(* Schneider Machine Expert - Basic project 撞击便携一体机, file version 1.5.0.0 *)
(* ProjectInformations: Name=New project *)

HARDWARE
  Cpu 0: TM200CE24U
  Cartridge1 0: TMCR2AM3
  EthernetConfiguration: NetworkName=M200, IpAllocationMode=FixedAddress, IpAddress=0.0.0.0, SubnetMask=0.0.0.0
  EthernetConfiguration: NetworkName=M221, IpAllocationMode=FixedAddress, IpAddress=0.0.0.0, SubnetMask=0.0.0.0
  SerialLineConfiguration: Baud=Baud19200, Parity=ParityEven, DataBits=DataBits8, StopBits=StopBits1, PhysicalMedium=PhysicalMediumRs485, TransmissionMode=TransmissionModeModbusRtu, SlaveId=1, Addressing=SlaveAddressing
  MastTask: UsePeriodScanMode=false, PeriodScan=2
  FastTask: Period=255
  CpuBehavior: StartingMode=StartAsPreviousState, AutoSaveRamOnEeprom=true, WatchdogPeriod=250

SYMBOLS  (address, symbol, comment, settings)
  %M0         "步进电机使能"
  %M1         "步进电机就位"
  %M2         "步进电机正向限位"
  %M3         "步进电机反向限位"
  %M4         "自动升锤任务表启动"
  %M5         "自动升锤任务表循环执行"
  %M6         "自动升锤任务表暂停执行"
  %M7         "装药任务表启动"
  %M8         "装药任务表循环执行"
  %M9         "装药任务表暂停执行"
  %M10        "吸放重锤电磁铁得电指令"
  %M11        "吸放重锤电磁铁失电指令"
  %M12        "自动降锤任务表启动"
  %M13        "落锤运动停止"
  %M15        "步进电机指令复位"
  %M16        "落锤运动模式(自动=1,手动=0)"
  %M17        "手动升锤"
  %M18        "手动降锤"
  %M19        "步进电机复位后n秒"
  %M20        "加压电机后退指令"
  %M21        "加压电机前进指令"
  %M22        "加压电机停止指令"
  %M23        "步进电机报警状态位"
  %M24        "系统复位"
  %M25        "撞击摩擦控制工艺区分位"
  %M26        "装药加压电机后退末程"
  %M30        "上位机重锤释放指令"
  %M31        "加压完成"
  %M32        "压力传感器开始受压时"
  %M33        "压力值接近设定压力时"
  %M34        "上位机装药指令"
  %M35        "靠近落锤位"
  %M36        "到达最低位"
  %M37        "到达装药位"
  %M38        "装药完成"
  %M39        "落锤运动方向位"
  %M40        "落锤向上减速位"
  %M41        "落锤向下减速位"
  %M42        "落锤向上运动到位"
  %M43        "落锤向下运动到位"
  %M45        "落锤运动到位"
  %M46        "落锤释放完成"
  %S13      SB_FIRSTRUN  "Indicates the first controller cycle in RUN mode"
  %MW1        "重锤位移中间原始值"
  %MW2        "重锤位移数字量差值"
  %MW3        "加压压力中间原始值"
  %MW4        "加压压力数字量差值"
  %MW5        "上位机落锤高度设置值(精确度：0.1mm)"
  %MW6        "上位机加压压力设置值(精确度:0.01T)"
  %MW7        "上位机重锤高度显示值（精确度：0.1mm)"
  %MW8        "上位机加压压力显示值(精确度:0.01T)"
  %MW9        "重锤运动量程值(精确度：0.1mm)"
  %MW10       "上位机高度显示中间值"
  %MW12       "上位机压力显示中间值"
  %MW15       "加压压力实数差值"
  %MW17       "加压压力实际实数值(单位:T)"
  %MW19       "重锤运动量程中间值"
  %MW21       "重锤位移实数差值"
  %MW23       "重锤位移实际实数值"
  %MW25       "重锤运动量程值"
  %MW27       "重锤相对位移实数值"
  %MW30       "上位机加压设置中间值"
  %MW32       "上位机加压设置转换值"
  %MW34       "加压电机频率设置值"
  %MW36       "加压电机频率设置值与量程比值"
  %MW38       "加压电机频率设置值对应数字量差值"
  %MW40       "加压电机频率设置值对应数字量值"
  %MW42       "加压电机频率整数值"
  %MW45       "加压设定值靠近值"
  %MW47       "上位机高度设置中间值"
  %MW49       "上位机高度设置转换值"
  %MW51       "落锤上升减速位移值"
  %MW53       "落锤下降减速位移值"
  %MW55       "位移相对值"
  %TM0        [Type=TP, Preset=1, Base=OneSecond]
  %TM1        [Preset=15, Base=OneHundredMilliSeconds]
  %TM2        [Preset=10, Base=OneSecond]
  %TM3        [Preset=21, Base=OneSecond]
  %TM4        [Preset=1, Base=OneSecond]
  %TM5        [Type=TP, Preset=2, Base=OneSecond]
  %MC_MOTIONTASK_PTO0   "升锤"  [Axis(Value(PtoAxis=PTO0)), StartStep(Value(int=1)), EndStep(Value(int=3)), Table(Value(PtoMotionTaskTable=Mt0))]
  %MC_MOTIONTASK_PTO1   "装药"  [Axis(Value(PtoAxis=PTO0)), StartStep(Value(int=1)), EndStep(Value(int=5)), Table(Value(PtoMotionTaskTable=Mt1))]
  %MC_MOVEABS_PTO0 绝对位置任务  [Axis(Value(PtoAxis=None)), Position(Value(int=10000)), Velocity(Value(int=20000)), Acceleration(Value(int=1000)), Deceleration(Value(int=1000)), JerkRatio(Value(int=0)), BufferMode(Value(BufferMode=McAborting))]
  %MC_MOVEREL_PTO1 相对位置任务1  [Axis(Value(PtoAxis=None)), Distance(Value(int=10000)), Velocity(Value(int=320)), Acceleration(Value(int=30)), Deceleration(Value(int=30)), JerkRatio(Value(int=0)), BufferMode(Value(BufferMode=McAborting))]
  %MC_MOVEREL_PTO6   [Axis(Value(PtoAxis=PTO0)), Distance(Value(int=10000)), Velocity(Value(int=200)), Acceleration(Value(int=30)), Deceleration(Value(int=30)), JerkRatio(Value(int=0)), BufferMode(Value(BufferMode=McAborting))]
  %MC_MOVEREL_PTO7   [Axis(Value(PtoAxis=PTO0)), Distance(Value(int=-10000)), Velocity(Value(int=50)), Acceleration(Value(int=30)), Deceleration(Value(int=30)), JerkRatio(Value(int=0)), BufferMode(Value(BufferMode=McAborting))]
  %MC_MOVEREL_PTO8   [Axis(Value(PtoAxis=PTO0)), Distance(Value(int=10000)), Velocity(Value(int=50)), Acceleration(Value(int=30)), Deceleration(Value(int=30)), JerkRatio(Value(int=0)), BufferMode(Value(BufferMode=McAborting))]
  %MC_MOVEVEL_PTO0 速度任务  [Axis(Value(PtoAxis=None)), Velocity(Value(int=10000)), Acceleration(Value(int=100)), Deceleration(Value(int=1000)), JerkRatio(Value(int=0)), Direction(Value(Direction=McPositiveDirection)), BufferMode(Value(BufferMode=McAborting))]
  %MC_POWER_PTO0   [Axis(Value(PtoAxis=PTO0))]
  %MC_RESET_PTO0   [Axis(Value(PtoAxis=PTO0))]
  %MC_SETPOS_PTO0 位置设定  [Axis(Value(PtoAxis=None)), Position(Value(int=0))]
  %MC_STOP_PTO0   [Axis(Value(PtoAxis=PTO0)), Deceleration(Value(int=30)), JerkRatio(Value(int=0))]
  %MT0        "升锤"  [IsConfigured=true, MotionSteps(MotionStep(Step=12, Type=None, Next=Done, Delay=0), MotionStep(Step=11, Type=None, Next=Done, Delay=0), MotionStep(Step=10, Type=None, Next=Done, Delay=0), MotionStep(Step=1, Pto=%MC_MOVEREL_PTO0, Type=MoveRelative, Next=SwEvent, Delay=0, Event=%M40), MotionStep(Step=13, Type=None, Next=Done, Delay=0), MotionStep(Step=2, Pto=%MC_MOVEREL_PTO5, Type=MoveRelative, Next=]
  %MT1        "装药"  [IsConfigured=true, MotionSteps(MotionStep(Step=1, Pto=%MC_MOVEREL_PTO1, Type=MoveRelative, Next=SwEvent, Delay=0, Event=%M35), MotionStep(Step=3, Pto=%MC_HALT_PTO1, Type=Halt, Next=Delay, Delay=500), MotionStep(Step=4, Pto=%MC_MOVEREL_PTO4, Type=MoveRelative, Next=SwEvent, Delay=0, Event=%M37), MotionStep(Step=5, Pto=%MC_HALT_PTO3, Type=Halt, Next=Done, Delay=0), MotionStep(Step=6, Type=None, Next]
  %I0.0       "加压电机后退限位"
  %I0.1       "安全门开关"
  %Q0.0       "步进电机脉冲位"
  %Q0.1       "吸放重锤电磁铁"
  %Q0.2       "步进电机方向位"
  %Q0.3       "加压电机后退"
  %Q0.4       "加压电机前进"
  %IW0.100  重锤原始位移值  [Type=Type_4_20_mA, Scope=Scope_Normal, Minimum=4000, Maximum=20000]
  %IW0.101  加压原始压力值  [Type=Type_4_20_mA, Scope=Scope_Normal, Minimum=4000, Maximum=20000]
  %QW0.100  加压变频电机频率  [Type=Type_4_20_mA, Scope=Scope_Normal, Minimum=4000, Maximum=20000]

POU 步进电机
  (* SectionNumber=1, IsGrafcet=false *)

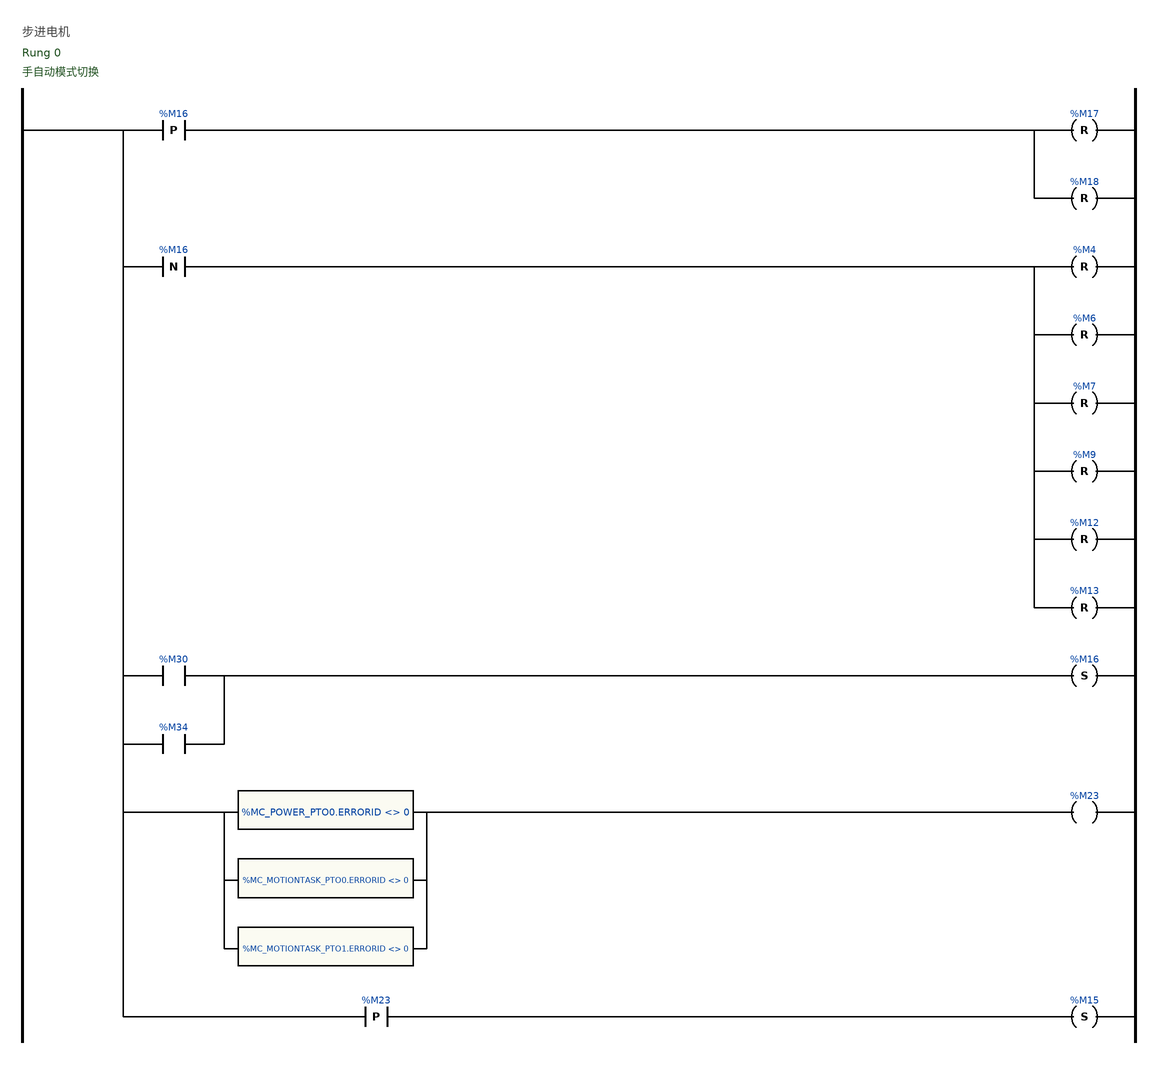

// Rung 0
// 手自动模式切换
  LD 1
  MPS
  ANDR %M16
  R %M17
  R %M18
  MRD
  ANDF %M16
  R %M4
  R %M6
  R %M7
  R %M9
  R %M12
  R %M13
  MRD
  AND( %M30
  OR %M34
  )
  S %M16
  MRD
  AND( [ %MC_POWER_PTO0.ERRORID <> 0 ]
  OR( [ %MC_MOTIONTASK_PTO0.ERRORID <> 0 ]
  OR [ %MC_MOTIONTASK_PTO1.ERRORID <> 0 ]
  )
  )
  ST %M23
  MPP
  ANDR %M23
  S %M15
  // as ST:
  //   IF RISING(%M16) THEN %M17 := FALSE; END_IF;
  //   IF RISING(%M16) THEN %M18 := FALSE; END_IF;
  //   IF FALLING(%M16) THEN %M4 := FALSE; END_IF;
  //   IF FALLING(%M16) THEN %M6 := FALSE; END_IF;
  //   IF FALLING(%M16) THEN %M7 := FALSE; END_IF;
  //   IF FALLING(%M16) THEN %M9 := FALSE; END_IF;
  //   IF FALLING(%M16) THEN %M12 := FALSE; END_IF;
  //   IF FALLING(%M16) THEN %M13 := FALSE; END_IF;
  //   IF %M30 OR %M34 THEN %M16 := TRUE; END_IF;
  //   %M23 := %MC_POWER_PTO0.ERRORID <> 0 OR %MC_MOTIONTASK_PTO0.ERRORID <> 0 OR %MC_MOTIONTASK_PTO1.ERRORID <> 0;
  //   IF RISING(%M23) THEN %M15 := TRUE; END_IF;

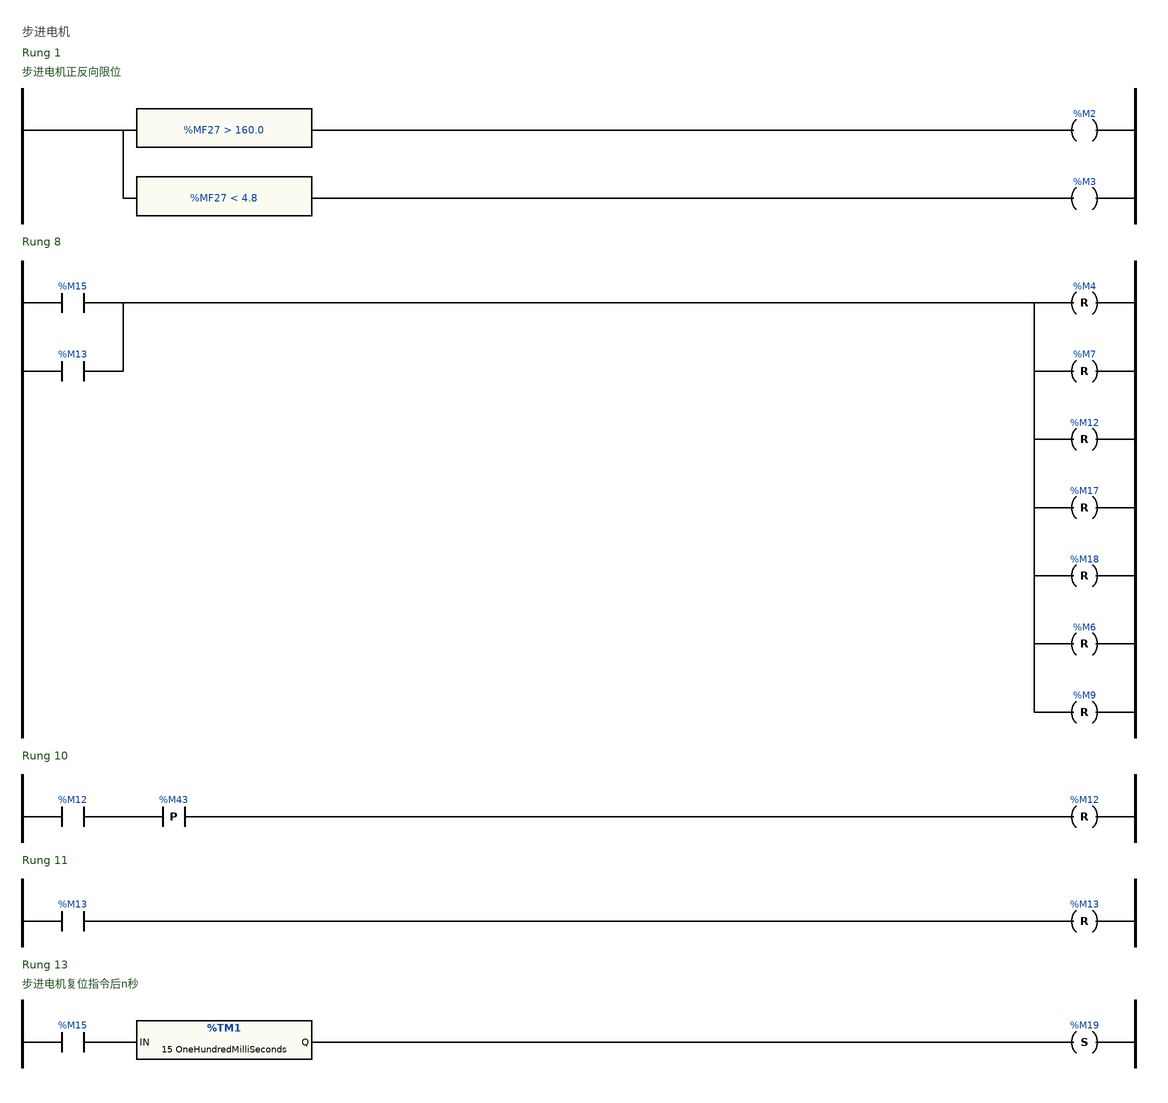

// Rung 1
// 步进电机正反向限位
  LD 1
  MPS
  AND [ %MF27 > 160.0 ]
  ST %M2
  MPP
  AND [ %MF27 < 4.8 ]
  ST %M3
  // as ST:
  //   %M2 := %MF27 > 160.0;
  //   %M3 := %MF27 < 4.8;

// Rung 2
// 步进电机使能及准备就位
  BLK %MC_POWER_PTO0
  LDN %M0
  Enable
  LDN %M1
  DriveReady
  LDN %M2
  OR %M15
  LimP
  LDN %M3
  OR %M15
  LimN
  END_BLK
  // as ST:
  //   %MC_POWER_PTO0(ENABLE := NOT %M0, DRIVEREADY := NOT %M1, LIMP := NOT %M2 OR %M15, LIMN := NOT %M3 OR %M15);
  (* the ladder stored for this rung does not match its IL; not drawn *)

// Rung 3
// 自动升锤
  BLK %MC_MOTIONTASK_PTO0
  LD %M4
  ANDN %M12
  ANDN %M7
  AND %M16
  Start
  LD %M5
  Loop
  LD %M6
  Pause
  OUT_BLK
  LD Ended
  R %M4
  END_BLK
  // as ST:
  //   %MC_MOTIONTASK_PTO0(START := %M4 AND NOT %M12 AND NOT %M7 AND %M16, LOOP := %M5, PAUSE := %M6);
  //   IF %MC_MOTIONTASK_PTO0.Ended THEN %M4 := FALSE; END_IF;
  (* the ladder stored for this rung does not match its IL; not drawn *)

// Rung 4
// 自动装药
  BLK %MC_MOTIONTASK_PTO1
  LD %M7
  ANDN %M4
  ANDN %M12
  AND %M16
  Start
  LD %M8
  Loop
  LD %M9
  Pause
  OUT_BLK
  LD Ended
  R %M7
  S %M38
  END_BLK
  // as ST:
  //   %MC_MOTIONTASK_PTO1(START := %M7 AND NOT %M4 AND NOT %M12 AND %M16, LOOP := %M8, PAUSE := %M9);
  //   IF %MC_MOTIONTASK_PTO1.Ended THEN %M7 := FALSE; END_IF;
  //   IF %MC_MOTIONTASK_PTO1.Ended THEN %M38 := TRUE; END_IF;
  (* the ladder stored for this rung does not match its IL; not drawn *)

// Rung 5
// 自动降锤
  BLK %MC_MOVEREL_PTO6
  LD %M12
  ANDN %M4
  ANDN %M7
  AND %M16
  Execute
  END_BLK
  // as ST:
  //   %MC_MOVEREL_PTO6(EXECUTE := %M12 AND NOT %M4 AND NOT %M7 AND %M16);
  (* the ladder stored for this rung does not match its IL; not drawn *)

// Rung 6
// 手动升锤
  BLK %MC_MOVEREL_PTO7
  LD %M17
  ANDN %M18
  ANDN %M16
  OR( %M19
  AND %M3
  )
  Execute
  END_BLK
  // as ST:
  //   %MC_MOVEREL_PTO7(EXECUTE := %M17 AND NOT %M18 AND NOT %M16 OR %M19 AND %M3);
  (* the ladder stored for this rung does not match its IL; not drawn *)

// Rung 7
// 手动降锤
  BLK %MC_MOVEREL_PTO8
  LD %M18
  ANDN %M17
  ANDN %M16
  OR( %M19
  AND %M2
  )
  Execute
  END_BLK
  // as ST:
  //   %MC_MOVEREL_PTO8(EXECUTE := %M18 AND NOT %M17 AND NOT %M16 OR %M19 AND %M2);
  (* the ladder stored for this rung does not match its IL; not drawn *)

// Rung 8
  LD %M15
  OR %M13
  R %M4
  R %M7
  R %M12
  R %M17
  R %M18
  R %M6
  R %M9
  // as ST:
  //   IF %M15 OR %M13 THEN %M4 := FALSE; END_IF;
  //   IF %M15 OR %M13 THEN %M7 := FALSE; END_IF;
  //   IF %M15 OR %M13 THEN %M12 := FALSE; END_IF;
  //   IF %M15 OR %M13 THEN %M17 := FALSE; END_IF;
  //   IF %M15 OR %M13 THEN %M18 := FALSE; END_IF;
  //   IF %M15 OR %M13 THEN %M6 := FALSE; END_IF;
  //   IF %M15 OR %M13 THEN %M9 := FALSE; END_IF;

// Rung 9
  BLK %MC_STOP_PTO0
  LD %M15
  OR( %M12
  ANDR %M43
  )
  OR %M13
  OR %M19
  Execute
  END_BLK
  // as ST:
  //   %MC_STOP_PTO0(EXECUTE := %M15 OR %M12 AND RISING(%M43) OR %M13 OR %M19);
  (* the ladder stored for this rung does not match its IL; not drawn *)

// Rung 10
  LD %M12
  ANDR %M43
  R %M12
  // as ST:
  //   IF %M12 AND RISING(%M43) THEN %M12 := FALSE; END_IF;

// Rung 11
  LD %M13
  R %M13
  // as ST:
  //   IF %M13 THEN %M13 := FALSE; END_IF;

// Rung 12
  BLK %MC_RESET_PTO0
  LD %M15
  Execute
  END_BLK
  // as ST:
  //   %MC_RESET_PTO0(EXECUTE := %M15);
  (* the ladder stored for this rung does not match its IL; not drawn *)

// Rung 13
// 步进电机复位指令后n秒
  BLK %TM1
  LD %M15
  IN
  OUT_BLK
  LD Q
  S %M19
  END_BLK
  // as ST:
  //   %TM1(IN := %M15);
  //   IF %TM1.Q THEN %M19 := TRUE; END_IF;

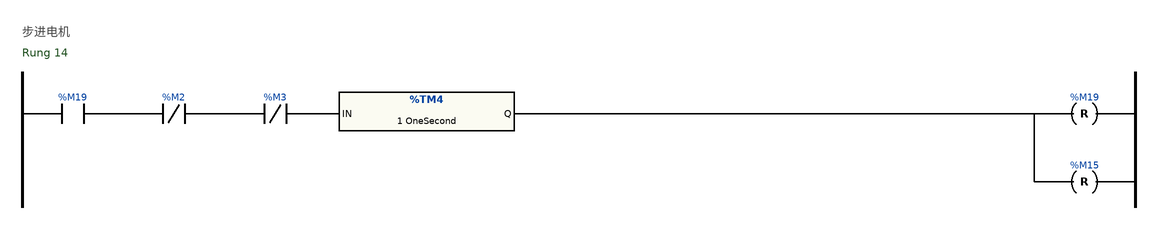

// Rung 14
  BLK %TM4
  LD %M19
  ANDN %M2
  ANDN %M3
  IN
  OUT_BLK
  LD Q
  R %M19
  R %M15
  END_BLK
  // as ST:
  //   %TM4(IN := %M19 AND NOT %M2 AND NOT %M3);
  //   IF %TM4.Q THEN %M19 := FALSE; END_IF;
  //   IF %TM4.Q THEN %M15 := FALSE; END_IF;

POU 吸放重锤电磁铁
  (* SectionNumber=2, IsGrafcet=false *)

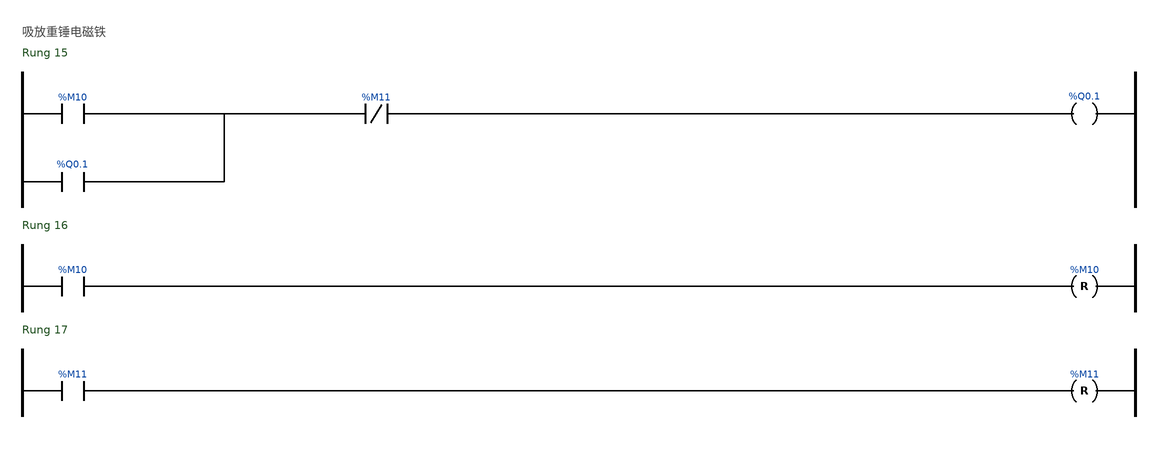

// Rung 15
  LD %M10
  OR %Q0.1
  ANDN %M11
  ST %Q0.1
  // as ST:
  //   %Q0.1 := (%M10 OR %Q0.1) AND NOT %M11;

// Rung 16
  LD %M10
  R %M10
  // as ST:
  //   IF %M10 THEN %M10 := FALSE; END_IF;

// Rung 17
  LD %M11
  R %M11
  // as ST:
  //   IF %M11 THEN %M11 := FALSE; END_IF;

POU 变频加压电机
  (* SectionNumber=3, IsGrafcet=false *)

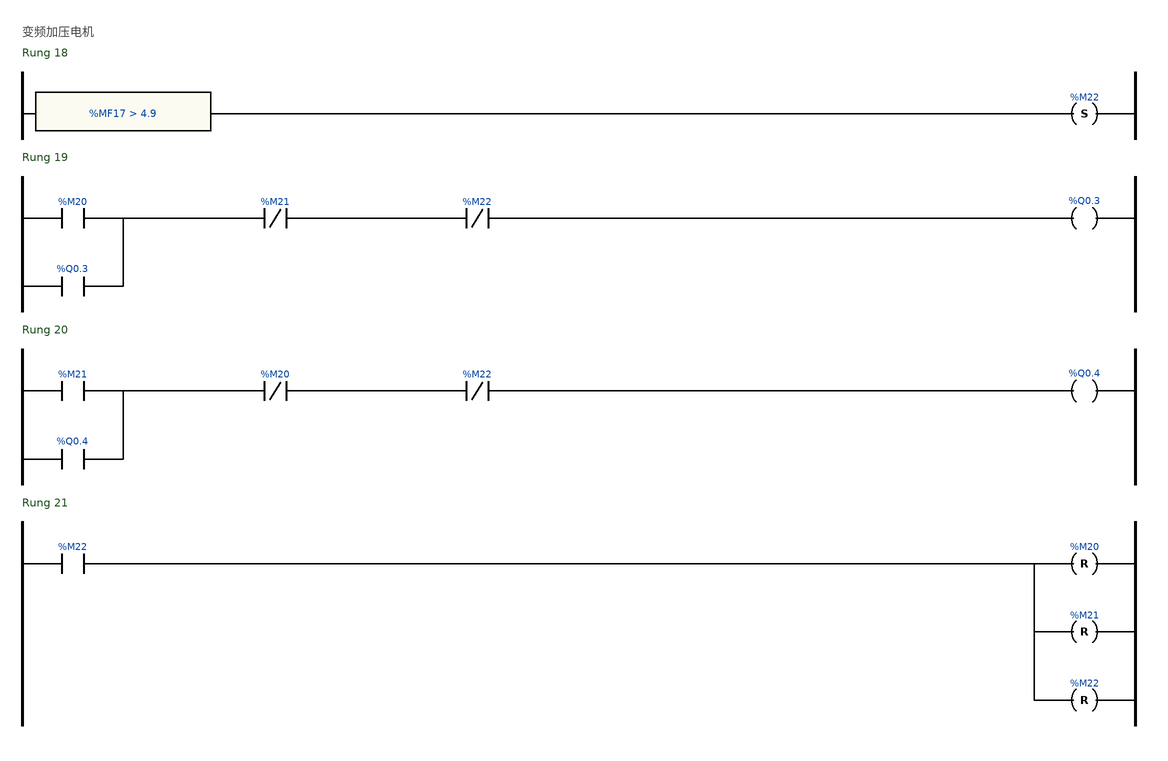

// Rung 18
  LD [ %MF17 > 4.9 ]
  S %M22
  // as ST:
  //   IF %MF17 > 4.9 THEN %M22 := TRUE; END_IF;

// Rung 19
  LD %M20
  OR %Q0.3
  ANDN %M21
  ANDN %M22
  ST %Q0.3
  // as ST:
  //   %Q0.3 := (%M20 OR %Q0.3) AND NOT %M21 AND NOT %M22;

// Rung 20
  LD %M21
  OR %Q0.4
  ANDN %M20
  ANDN %M22
  ST %Q0.4
  // as ST:
  //   %Q0.4 := (%M21 OR %Q0.4) AND NOT %M20 AND NOT %M22;

// Rung 21
  LD %M22
  R %M20
  R %M21
  R %M22
  // as ST:
  //   IF %M22 THEN %M20 := FALSE; END_IF;
  //   IF %M22 THEN %M21 := FALSE; END_IF;
  //   IF %M22 THEN %M22 := FALSE; END_IF;

POU 重锤位移值
  (* SectionNumber=4, IsGrafcet=false *)

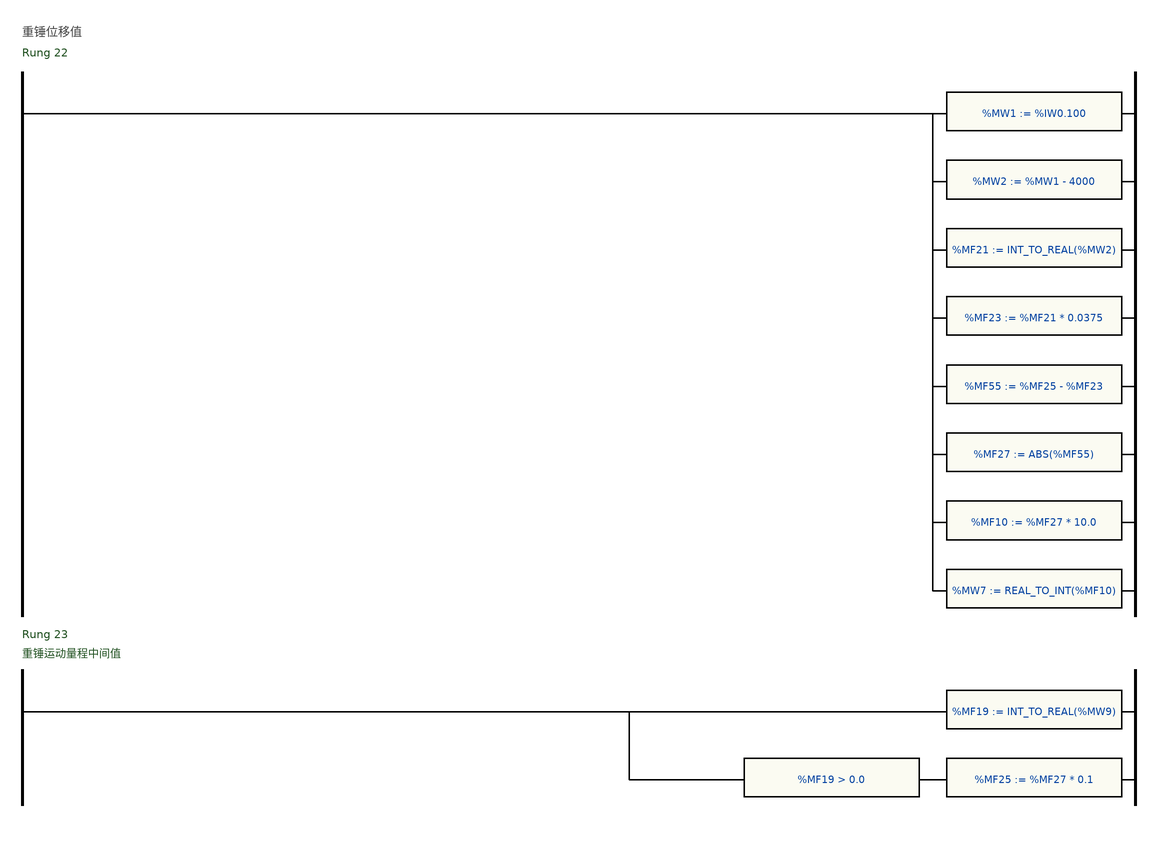

// Rung 22
  LD 1
  [ %MW1 := %IW0.100 ]    (* 重锤原始位移值 *)
  [ %MW2 := %MW1 - 4000 ]
  [ %MF21 := INT_TO_REAL ( %MW2 ) ]
  [ %MF23 := %MF21 * 0.0375 ]
  [ %MF55 := %MF25 - %MF23 ]
  [ %MF27 := ABS ( %MF55 ) ]
  [ %MF10 := %MF27 * 10.0 ]
  [ %MW7 := REAL_TO_INT ( %MF10 ) ]
  // as ST:
  //   %MW1 := 重锤原始位移值;
  //   %MW2 := %MW1 - 4000;
  //   %MF21 := INT_TO_REAL ( %MW2 );
  //   %MF23 := %MF21  *  0.0375;
  //   %MF55 := %MF25  -  %MF23;
  //   %MF27 := ABS ( %MF55 );
  //   %MF10 := %MF27  *  10.0;
  //   %MW7 := REAL_TO_INT ( %MF10 );

// Rung 23
// 重锤运动量程中间值
  LD 1
  MPS
  [ %MF19 := INT_TO_REAL ( %MW9 ) ]
  MPP
  AND [ %MF19 > 0.0 ]
  [ %MF25 := %MF27 * 0.1 ]
  // as ST:
  //   %MF19 := INT_TO_REAL ( %MW9 );
  //   IF %MF19 > 0.0 THEN %MF25 := %MF27  *  0.1; END_IF;

POU 加压压力值
  (* SectionNumber=5, IsGrafcet=false *)

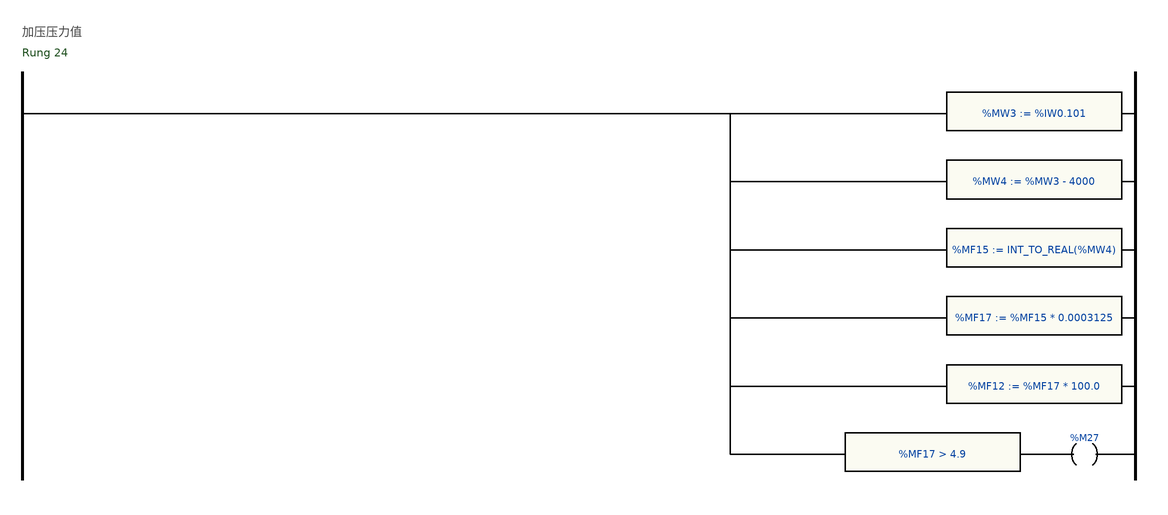

// Rung 24
  LD 1
  MPS
  [ %MW3 := %IW0.101 ]    (* 加压原始压力值 *)
  MRD
  [ %MW4 := %MW3 - 4000 ]
  MRD
  [ %MF15 := INT_TO_REAL ( %MW4 ) ]
  MRD
  [ %MF17 := %MF15 * 0.0003125 ]
  MRD
  [ %MF12 := %MF17 * 100.0 ]
  MPP
  AND [ %MF17 > 4.9 ]
  ST %M27
  // as ST:
  //   %MW3 := 加压原始压力值;
  //   %MW4 := %MW3 - 4000;
  //   %MF15 := INT_TO_REAL ( %MW4 );
  //   %MF17 := %MF15  *  0.0003125;
  //   %MF12 := %MF17  *  100.0;
  //   %M27 := %MF17 > 4.9;

POU 加压电机频率
  (* SectionNumber=6, IsGrafcet=false *)

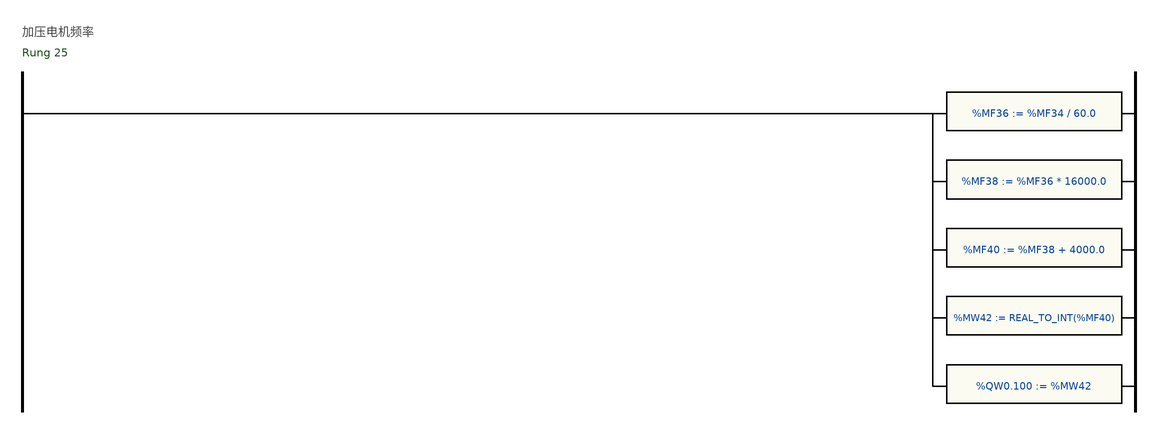

// Rung 25
  LD 1
  [ %MF36 := %MF34 / 60.0 ]
  [ %MF38 := %MF36 * 16000.0 ]
  [ %MF40 := %MF38 + 4000.0 ]
  [ %MW42 := REAL_TO_INT ( %MF40 ) ]
  [ %QW0.100 := %MW42 ]   (* 加压变频电机频率 *)
  // as ST:
  //   %MF36 := %MF34  /  60.0;
  //   %MF38 := %MF36  *  16000.0;
  //   %MF40 := %MF38  +  4000.0;
  //   %MW42 := REAL_TO_INT ( %MF40 );
  //   加压变频电机频率 := %MW42;

POU 加压逻辑
  (* SectionNumber=7, IsGrafcet=false *)

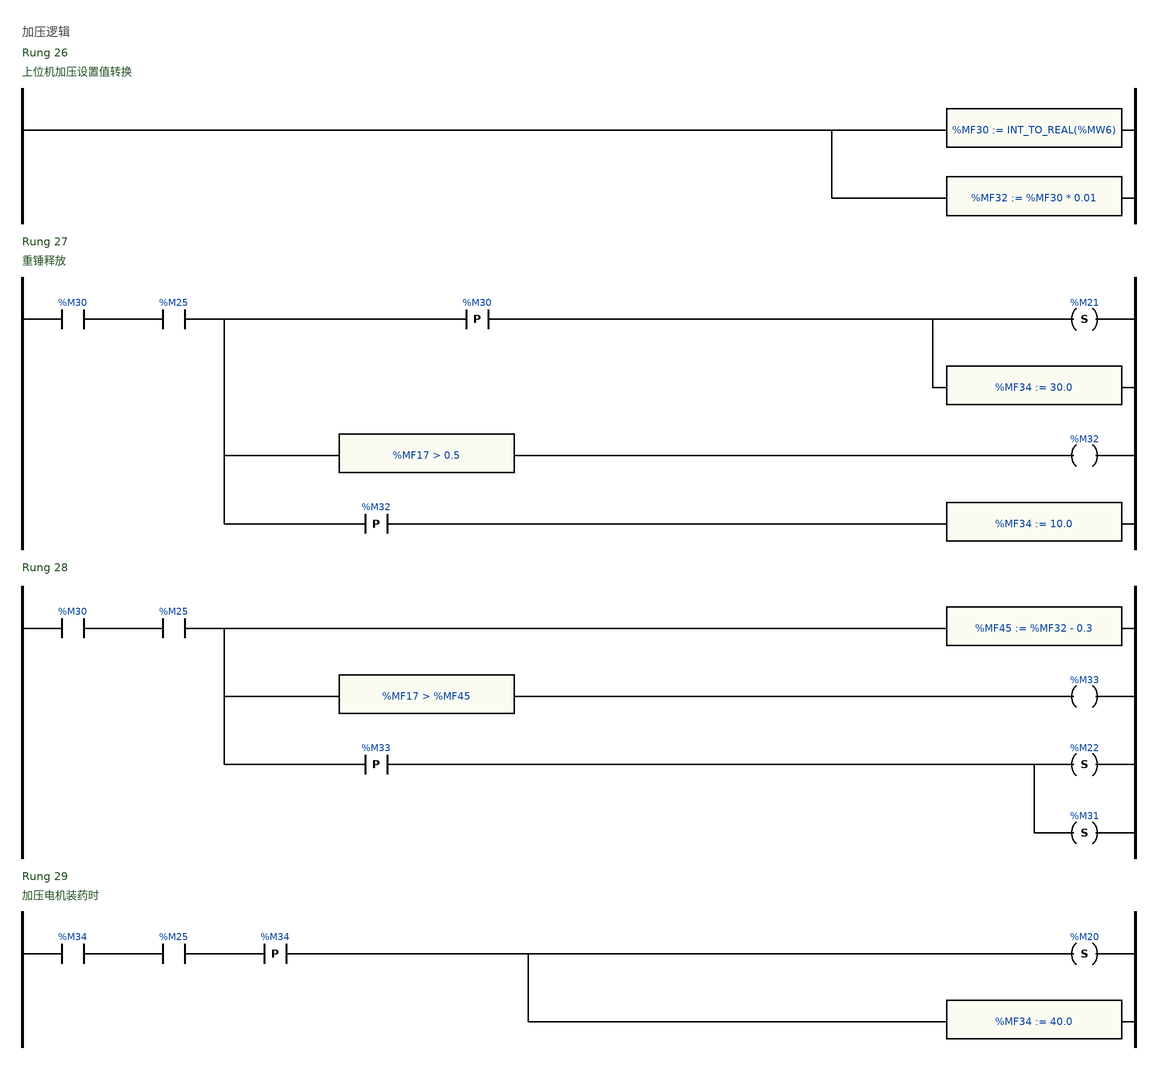

// Rung 26
// 上位机加压设置值转换
  LD 1
  [ %MF30 := INT_TO_REAL ( %MW6 ) ]
  [ %MF32 := %MF30 * 0.01 ]
  // as ST:
  //   %MF30 := INT_TO_REAL ( %MW6 );
  //   %MF32 := %MF30  *  0.01;

// Rung 27
// 重锤释放
  LD %M30
  AND %M25
  MPS
  ANDR %M30
  S %M21
  [ %MF34 := 30.0 ]
  MRD
  AND [ %MF17 > 0.5 ]
  ST %M32
  MPP
  ANDR %M32
  [ %MF34 := 10.0 ]
  // as ST:
  //   IF %M30 AND %M25 AND RISING(%M30) THEN %M21 := TRUE; END_IF;
  //   IF %M30 AND %M25 AND RISING(%M30) THEN %MF34 := 30.0; END_IF;
  //   %M32 := %M30 AND %M25 AND %MF17 > 0.5;
  //   IF %M30 AND %M25 AND RISING(%M32) THEN %MF34 := 10.0; END_IF;

// Rung 28
  LD %M30
  AND %M25
  MPS
  [ %MF45 := %MF32 - 0.3 ]
  MRD
  AND [ %MF17 > %MF45 ]
  ST %M33
  MPP
  ANDR %M33
  S %M22
  S %M31
  // as ST:
  //   IF %M30 AND %M25 THEN %MF45 := %MF32  -  0.3; END_IF;
  //   %M33 := %M30 AND %M25 AND %MF17 > %MF45;
  //   IF %M30 AND %M25 AND RISING(%M33) THEN %M22 := TRUE; END_IF;
  //   IF %M30 AND %M25 AND RISING(%M33) THEN %M31 := TRUE; END_IF;

// Rung 29
// 加压电机装药时
  LD %M34
  AND %M25
  ANDR %M34
  S %M20
  [ %MF34 := 40.0 ]
  // as ST:
  //   IF %M34 AND %M25 AND RISING(%M34) THEN %M20 := TRUE; END_IF;
  //   IF %M34 AND %M25 AND RISING(%M34) THEN %MF34 := 40.0; END_IF;

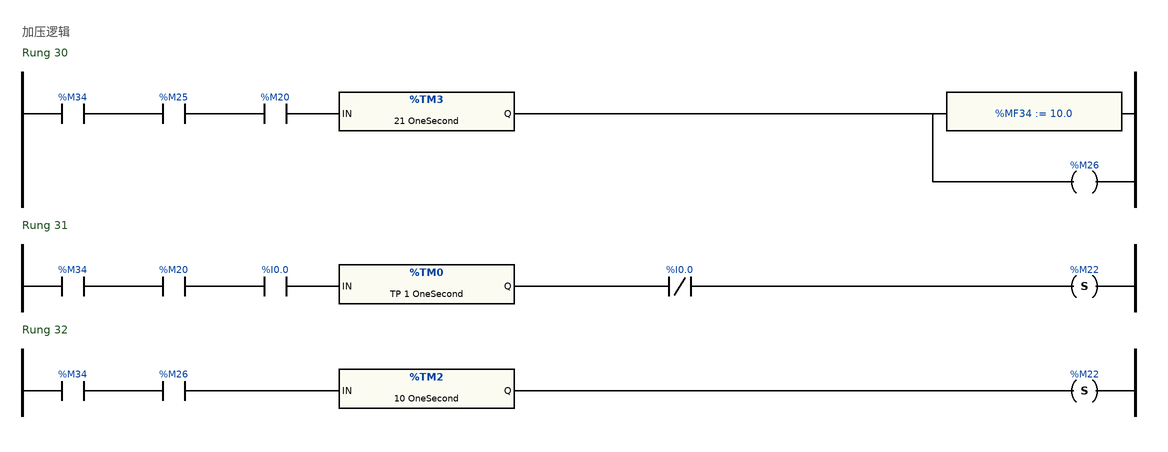

// Rung 30
  BLK %TM3
  LD %M34
  AND %M25
  AND %M20
  IN
  OUT_BLK
  LD Q
  [ %MF34 := 10.0 ]
  ST %M26
  END_BLK
  // as ST:
  //   %TM3(IN := %M34 AND %M25 AND %M20);
  //   IF %TM3.Q THEN %MF34 := 10.0; END_IF;
  //   %M26 := %TM3.Q;

// Rung 31
  BLK %TM0
  LD %M34
  AND %M20
  AND %I0.0
  IN
  OUT_BLK
  LD Q
  ANDN %I0.0
  S %M22
  END_BLK
  // as ST:
  //   %TM0(IN := %M34 AND %M20 AND %I0.0);
  //   IF %TM0.Q AND NOT %I0.0 THEN %M22 := TRUE; END_IF;

// Rung 32
  BLK %TM2
  LD %M34
  AND %M26
  IN
  OUT_BLK
  LD Q
  S %M22
  END_BLK
  // as ST:
  //   %TM2(IN := %M34 AND %M26);
  //   IF %TM2.Q THEN %M22 := TRUE; END_IF;

POU 装药/放锤
  (* SectionNumber=8, IsGrafcet=false *)

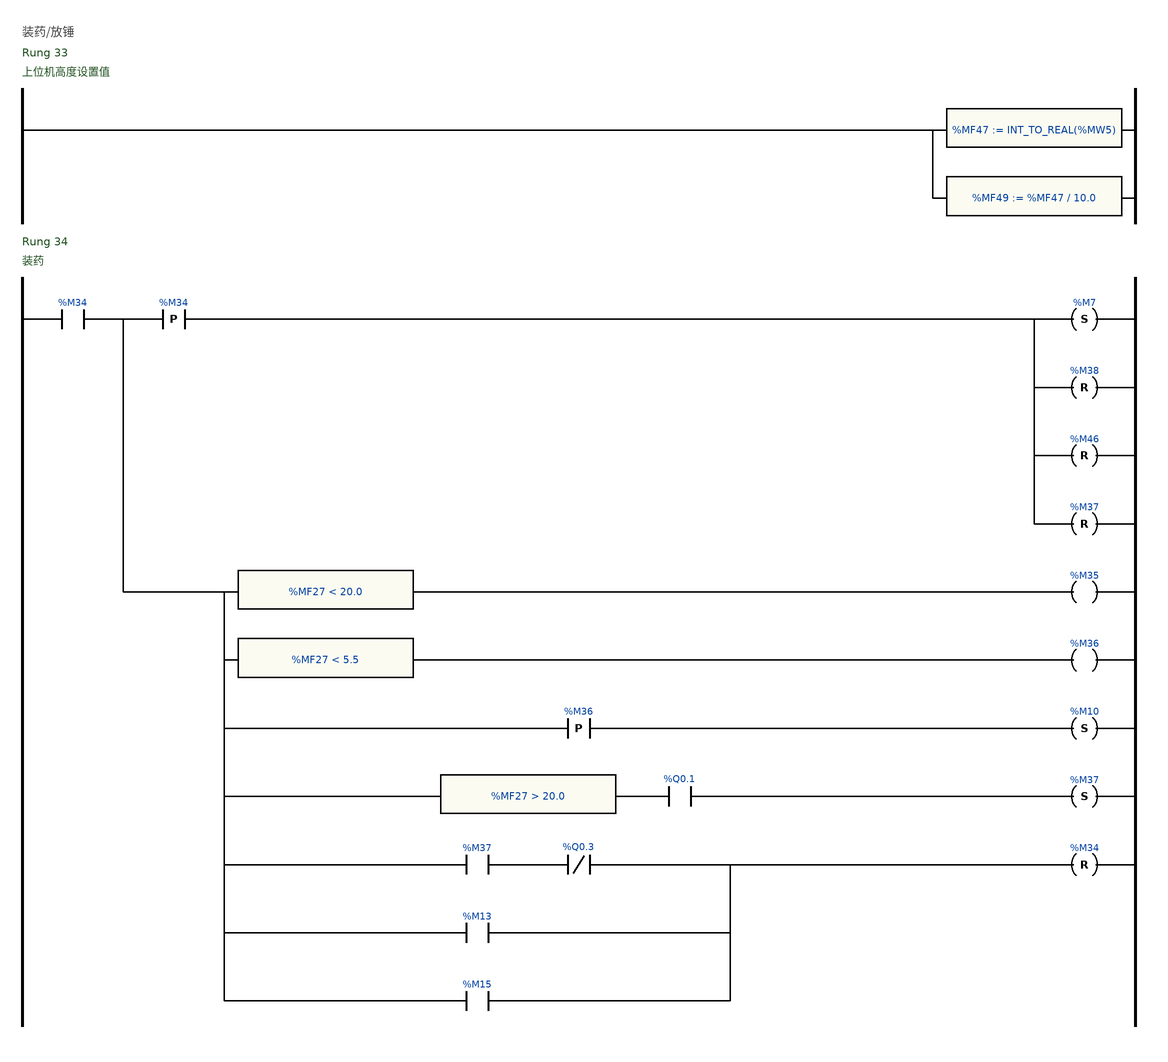

// Rung 33
// 上位机高度设置值
  LD 1
  [ %MF47 := INT_TO_REAL ( %MW5 ) ]
  [ %MF49 := %MF47 / 10.0 ]
  // as ST:
  //   %MF47 := INT_TO_REAL ( %MW5 );
  //   %MF49 := %MF47  /  10.0;

// Rung 34
// 装药
  LD %M34
  MPS
  ANDR %M34
  S %M7
  R %M38
  R %M46
  R %M37
  MRD
  AND [ %MF27 < 20.0 ]
  ST %M35
  MRD
  AND [ %MF27 < 5.5 ]
  ST %M36
  MRD
  ANDR %M36
  S %M10
  MRD
  AND [ %MF27 > 20.0 ]
  AND %Q0.1
  S %M37
  MPP
  AND( %M37
  ANDN %Q0.3
  OR %M13
  OR %M15
  )
  R %M34
  // as ST:
  //   IF %M34 AND RISING(%M34) THEN %M7 := TRUE; END_IF;
  //   IF %M34 AND RISING(%M34) THEN %M38 := FALSE; END_IF;
  //   IF %M34 AND RISING(%M34) THEN %M46 := FALSE; END_IF;
  //   IF %M34 AND RISING(%M34) THEN %M37 := FALSE; END_IF;
  //   %M35 := %M34 AND %MF27 < 20.0;
  //   %M36 := %M34 AND %MF27 < 5.5;
  //   IF %M34 AND RISING(%M36) THEN %M10 := TRUE; END_IF;
  //   IF %M34 AND %MF27 > 20.0 AND %Q0.1 THEN %M37 := TRUE; END_IF;
  //   IF %M34 AND (%M37 AND NOT %Q0.3 OR %M13 OR %M15) THEN %M34 := FALSE; END_IF;

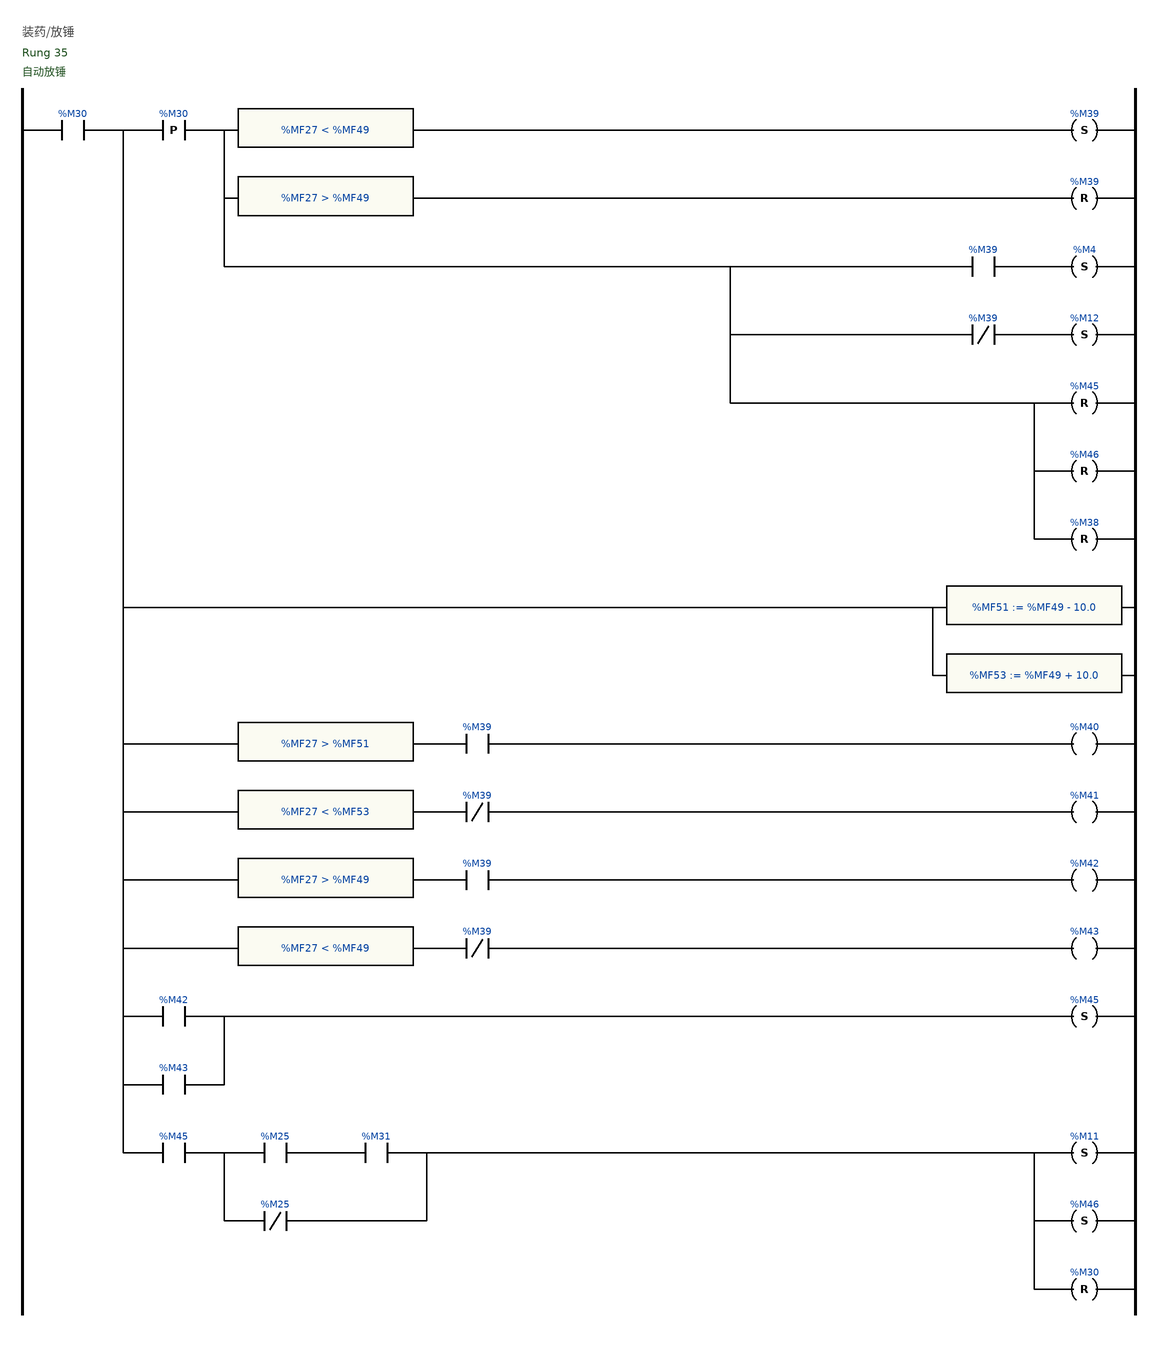

// Rung 35
// 自动放锤
  LD %M30
  MPS
  ANDR %M30
  MPS
  AND [ %MF27 < %MF49 ]
  S %M39
  MRD
  AND [ %MF27 > %MF49 ]
  R %M39
  MRD
  AND %M39
  S %M4
  MRD
  ANDN %M39
  S %M12
  MPP
  R %M45
  R %M46
  R %M38
  MRD
  [ %MF51 := %MF49 - 10.0 ]
  [ %MF53 := %MF49 + 10.0 ]
  MRD
  AND [ %MF27 > %MF51 ]
  AND %M39
  ST %M40
  MRD
  AND [ %MF27 < %MF53 ]
  ANDN %M39
  ST %M41
  MRD
  AND [ %MF27 > %MF49 ]
  AND %M39
  ST %M42
  MRD
  AND [ %MF27 < %MF49 ]
  ANDN %M39
  ST %M43
  MRD
  AND( %M42
  OR %M43
  )
  S %M45
  MPP
  AND %M45
  AND( %M25
  AND %M31
  ORN %M25
  )
  S %M11
  S %M46
  R %M30
  // as ST:
  //   IF %M30 AND RISING(%M30) AND %MF27 < %MF49 THEN %M39 := TRUE; END_IF;
  //   IF %M30 AND RISING(%M30) AND %MF27 > %MF49 THEN %M39 := FALSE; END_IF;
  //   IF %M30 AND RISING(%M30) AND %M39 THEN %M4 := TRUE; END_IF;
  //   IF %M30 AND RISING(%M30) AND NOT %M39 THEN %M12 := TRUE; END_IF;
  //   IF %M30 AND RISING(%M30) THEN %M45 := FALSE; END_IF;
  //   IF %M30 AND RISING(%M30) THEN %M46 := FALSE; END_IF;
  //   IF %M30 AND RISING(%M30) THEN %M38 := FALSE; END_IF;
  //   IF %M30 THEN %MF51 := %MF49  -  10.0; END_IF;
  //   IF %M30 THEN %MF53 := %MF49  +  10.0; END_IF;
  //   %M40 := %M30 AND %MF27 > %MF51 AND %M39;
  //   %M41 := %M30 AND %MF27 < %MF53 AND NOT %M39;
  //   %M42 := %M30 AND %MF27 > %MF49 AND %M39;
  //   %M43 := %M30 AND %MF27 < %MF49 AND NOT %M39;
  //   IF %M30 AND (%M42 OR %M43) THEN %M45 := TRUE; END_IF;
  //   IF %M30 AND %M45 AND (%M25 AND %M31 OR NOT %M25) THEN %M11 := TRUE; END_IF;
  //   IF %M30 AND %M45 AND (%M25 AND %M31 OR NOT %M25) THEN %M46 := TRUE; END_IF;
  //   IF %M30 AND %M45 AND (%M25 AND %M31 OR NOT %M25) THEN %M30 := FALSE; END_IF;

POU 初始化
  (* SectionNumber=9, IsGrafcet=false *)

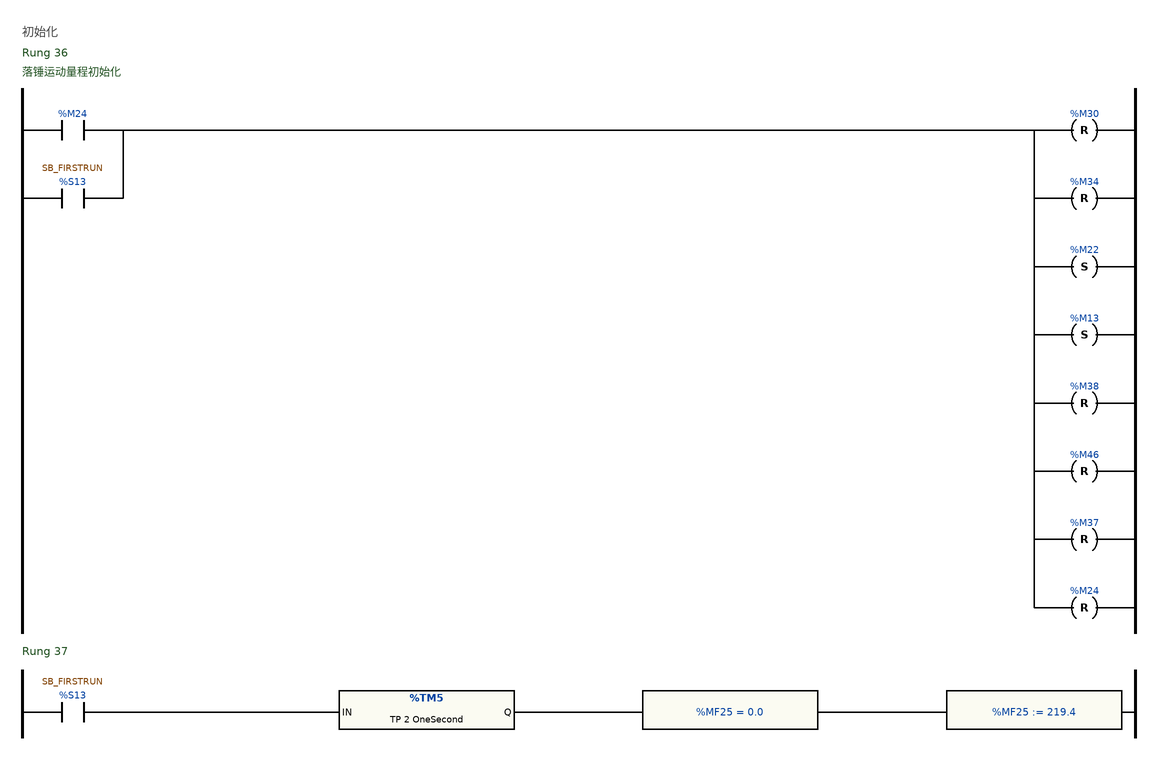

// Rung 36
// 落锤运动量程初始化
  LD %M24
  OR %S13                 (* SB_FIRSTRUN *)
  R %M30
  R %M34
  S %M22
  S %M13
  R %M38
  R %M46
  R %M37
  R %M24
  // as ST:
  //   IF %M24 OR SB_FIRSTRUN THEN %M30 := FALSE; END_IF;
  //   IF %M24 OR SB_FIRSTRUN THEN %M34 := FALSE; END_IF;
  //   IF %M24 OR SB_FIRSTRUN THEN %M22 := TRUE; END_IF;
  //   IF %M24 OR SB_FIRSTRUN THEN %M13 := TRUE; END_IF;
  //   IF %M24 OR SB_FIRSTRUN THEN %M38 := FALSE; END_IF;
  //   IF %M24 OR SB_FIRSTRUN THEN %M46 := FALSE; END_IF;
  //   IF %M24 OR SB_FIRSTRUN THEN %M37 := FALSE; END_IF;
  //   IF %M24 OR SB_FIRSTRUN THEN %M24 := FALSE; END_IF;

// Rung 37
  BLK %TM5
  LD %S13                 (* SB_FIRSTRUN *)
  IN
  OUT_BLK
  LD Q
  AND [ %MF25 = 0.0 ]
  [ %MF25 := 219.4 ]
  END_BLK
  // as ST:
  //   %TM5(IN := SB_FIRSTRUN);
  //   IF %TM5.Q AND %MF25 = 0.0 THEN %MF25 := 219.4; END_IF;
